(* IEC 61131-3 sources: simulador/simulador_codesys, 11 files *)

(* ---- GVL_SimConfig.st ---- *)
// =============================================================================
// GVL_SimConfig — Parâmetros globais de configuração do simulador
// Equivalente a: config.py + config_etapa1/2/3.yaml
//
// COMO USAR:
//   Etapa 1 (loopback)  → SIM_MODE := 0
//   Etapa 2 (openloop)  → SIM_MODE := 1
//   Etapa 3 (full)      → SIM_MODE := 2
//
// Alterar SIM_MODE em tempo de execução reinicializa o comportamento na
// próxima chamada de FB_Simulator (bEdgeInit detecta a mudança).
// =============================================================================

VAR_GLOBAL CONSTANT

    // -------------------------------------------------------------------------
    // Modo de simulação
    //   0 = LOOPBACK  — comunicação Modbus, medidor fixo, física OFF
    //   1 = OPENLOOP  — física ON, carga/irradiância fixas, sem perfis/eventos
    //   2 = FULL      — física ON, perfis ativos, eventos ativos
    // -------------------------------------------------------------------------
    SIM_MODE_LOOPBACK   : INT := 0;
    SIM_MODE_OPENLOOP   : INT := 1;
    SIM_MODE_FULL       : INT := 2;

    // -------------------------------------------------------------------------
    // Temporização
    // -------------------------------------------------------------------------
    TICK_S              : REAL := 0.05;     // Período do ciclo de simulação (s)
                                             // Deve coincidir com o período da
                                             // task cíclica no Codesys Scheduler.
                                             // 50 ms é o mínimo seguro.

    // -------------------------------------------------------------------------
    // Rede elétrica
    // -------------------------------------------------------------------------
    V_LL_V              : REAL := 380.0;    // Tensão nominal linha-linha BT (V)
    V_MT_LL_V           : REAL := 13800.0;  // Tensão nominal linha-linha MT (V)

    // -------------------------------------------------------------------------
    // Equivalente de Thévenin da rede (referido ao BT)
    // -------------------------------------------------------------------------
    THEVENIN_VTH_LL_V   : REAL := 380.0;   // Tensão de Thévenin LL (V)
    THEVENIN_R_OHM      : REAL := 0.00283; // Resistência equivalente (Ω)
    THEVENIN_X_OHM      : REAL := 0.01416; // Reatância equivalente (Ω)

    // -------------------------------------------------------------------------
    // Relações de transformação dos instrumentos
    // -------------------------------------------------------------------------
    RTP                 : REAL := 120.0;    // Relação do TP  (ex: 13800/115 → 120)
    RTC                 : REAL := 200.0;    // Relação do TC  (ex: 200/5 → 200)

    // -------------------------------------------------------------------------
    // Modelo de carga ZIP (coeficientes ANEEL para alimentadores)
    //   P: 50% impedância constante + 50% potência constante
    //   Q: 100% potência constante
    // -------------------------------------------------------------------------
    ZIP_P_Z             : REAL := 0.50;    // Fração Z para P
    ZIP_P_I             : REAL := 0.00;    // Fração I para P
    ZIP_P_P             : REAL := 0.50;    // Fração P para P
    ZIP_Q_Z             : REAL := 0.00;    // Fração Z para Q
    ZIP_Q_I             : REAL := 0.00;    // Fração I para Q
    ZIP_Q_P             : REAL := 1.00;    // Fração P para Q

    // -------------------------------------------------------------------------
    // Carga padrão (usada em openloop e como fallback no full)
    // -------------------------------------------------------------------------
    LOAD_P_KW_DEFAULT   : REAL := 200.0;   // Potência ativa da carga (kW)
    LOAD_Q_KVAR_DEFAULT : REAL := 50.0;    // Potência reativa da carga (kVAr)

    // -------------------------------------------------------------------------
    // Irradiância padrão (normalizada 0.0..1.0)
    // -------------------------------------------------------------------------
    U_DEFAULT           : REAL := 1.0;     // 1.0 = irradiância plena (100%)

    // -------------------------------------------------------------------------
    // Valores fixos do medidor no modo LOOPBACK (grandezas no SECUNDÁRIO)
    //   V_sec_fn = V_MT_fn / RTP = (13800 / sqrt(3)) / 120 ≈ 66.4 V
    //   I_sec    = valor de teste no secundário do TC
    //   PF       = fator de potência de teste
    // -------------------------------------------------------------------------
    LOOPBACK_PF         : REAL := 0.92;    // Fator de potência fixo (loopback)
    LOOPBACK_V_MT_LN_V  : REAL := 66.4;   // Tensão sec. TP fase-neutro (V)
    LOOPBACK_I_MT_A     : REAL := 2.5;    // Corrente sec. TC (A)

    // -------------------------------------------------------------------------
    // Medidor Modbus (slave 100, COM1)
    // -------------------------------------------------------------------------
    METER_SLAVE_ID      : INT  := 100;
    METER_BASE_ADDR     : INT  := 153;     // 0x0099 decimal — endereço base FC03
    METER_QTY_U16       : INT  := 28;      // Quantidade de registradores U16

    // -------------------------------------------------------------------------
    // Número total de inversores
    //   COM1: slaves 101..109  (9 inversores)
    //   COM2: slaves 201..209  (9 inversores)
    // -------------------------------------------------------------------------
    N_INV               : INT  := 18;      // Total de inversores
    N_INV_COM1          : INT  := 9;       // Inversores na COM1 (índices 0..8)
    N_INV_COM2          : INT  := 9;       // Inversores na COM2 (índices 9..17)

    // -------------------------------------------------------------------------
    // Slave IDs dos inversores
    //   Índice 0..8  → COM1: slaves 101..109
    //   Índice 9..17 → COM2: slaves 201..209
    // -------------------------------------------------------------------------
    INV_SLAVE_ID        : ARRAY[0..17] OF INT := [
        101, 102, 103, 104, 105, 106, 107, 108, 109,   // COM1
        201, 202, 203, 204, 205, 206, 207, 208, 209    // COM2
    ];

    // -------------------------------------------------------------------------
    // Potências nominais dos inversores (kW)
    // -------------------------------------------------------------------------
    INV_P_NOM_KW        : ARRAY[0..17] OF REAL := [
        60.0, 60.0, 35.0, 15.0, 15.0, 15.0, 15.0, 15.0, 15.0,  // COM1
        15.0, 15.0, 15.0, 15.0, 15.0, 15.0, 35.0, 35.0, 50.0   // COM2
    ];

    // -------------------------------------------------------------------------
    // Potências aparentes nominais dos inversores (kVA)
    // -------------------------------------------------------------------------
    INV_S_NOM_KVA       : ARRAY[0..17] OF REAL := [
        60.0, 60.0, 35.0, 15.0, 15.0, 15.0, 15.0, 15.0, 15.0,  // COM1
        15.0, 15.0, 15.0, 15.0, 15.0, 15.0, 35.0, 35.0, 50.0   // COM2
    ];

    // -------------------------------------------------------------------------
    // Constantes de tempo dos inversores (s)
    //   tau_p: dinâmica de P (1ª ordem)
    //   tau_q: dinâmica de Q (1ª ordem)
    // -------------------------------------------------------------------------
    INV_TAU_P_S         : ARRAY[0..17] OF REAL := [
        1.0, 1.0, 1.0, 1.0, 1.0, 1.0, 1.0, 1.0, 1.0,
        1.0, 1.0, 1.0, 1.0, 1.0, 1.0, 1.0, 1.0, 1.0
    ];
    INV_TAU_Q_S         : ARRAY[0..17] OF REAL := [
        1.0, 1.0, 1.0, 1.0, 1.0, 1.0, 1.0, 1.0, 1.0,
        1.0, 1.0, 1.0, 1.0, 1.0, 1.0, 1.0, 1.0, 1.0
    ];

    // -------------------------------------------------------------------------
    // Endereços Modbus dos inversores (Holding Registers, base 0)
    // -------------------------------------------------------------------------
    INV_HR_P_PCT        : INT := 256;      // HR 256 → setpoint %P  (escrito pelo master)
    INV_HR_PF_RAW       : INT := 257;      // HR 257 → FP raw       (escrito pelo master)

    // -------------------------------------------------------------------------
    // Eventos: intervalo de releitura (s)
    // -------------------------------------------------------------------------
    EVENTS_POLL_S       : REAL := 2.0;

END_VAR

(* ---- GVL_SimState.st ---- *)
// =============================================================================
// GVL_SimState — Estado em tempo de execução do simulador
// Equivalente às dataclasses InverterState, MeterState e PlantSimulation
// em simulation.py.
//
// Estas variáveis são LIDAS/ESCRITAS pelo FB_Simulator a cada ciclo.
// O driver Modbus Slave do Codesys mapeia diretamente os registradores
// do medidor (MW_Meter) e dos inversores (MW_Inv_*) em memória.
// =============================================================================

VAR_GLOBAL

    // =========================================================================
    // CONTROLE GERAL
    // =========================================================================

    // Modo ativo (alterável em runtime via HMI ou variável)
    //   0 = LOOPBACK | 1 = OPENLOOP | 2 = FULL
    g_SimMode           : INT := 0;

    // Tempo acumulado de simulação (s) — avança a cada ciclo
    g_T_s               : REAL := 0.0;

    // Flag de reinicialização: setar TRUE para reiniciar estados
    g_Reset             : BOOL := FALSE;

    // =========================================================================
    // ESTADO DOS INVERSORES
    // =========================================================================

    // --- Setpoints recebidos do master via FC16 (escritos pelo driver Modbus) ---
    // HR 256: setpoint %P  (0..100)
    g_Inv_P_Ref_Pct     : ARRAY[0..17] OF REAL := [18(0.0)];

    // HR 257: FP raw (1..100)
    g_Inv_PF_Cmd_Raw    : ARRAY[0..17] OF INT  := [18(100)];

    // --- Estados internos da dinâmica de 1ª ordem ---
    g_Inv_P_kW          : ARRAY[0..17] OF REAL := [18(0.0)];
    g_Inv_Q_kVAr        : ARRAY[0..17] OF REAL := [18(0.0)];

    // --- Disponibilidade de energia (irradiância normalizada 0..1) ---
    g_Inv_U             : ARRAY[0..17] OF REAL := [18(1.0)];

    // --- Flags de eventos ---
    g_Inv_CommsDrop     : ARRAY[0..17] OF BOOL := [18(FALSE)];
    g_Inv_Frozen_s      : ARRAY[0..17] OF REAL := [18(0.0)];

    // =========================================================================
    // ESTADO DO MEDIDOR (grandezas no SECUNDÁRIO dos instrumentos)
    // =========================================================================
    // O driver Modbus Slave mapeia MW_Meter[] nos registradores FC03
    // a partir do endereço base 0x0099 (153 decimal).
    // Cada elemento é um UINT (U16) codificado conforme especificação.

    // Registradores raw U16 para o driver Modbus Slave
    // Índice 0..27 → offsets relativos a 0x0099
    //   [0]  = PF fase A     [1]  = PF fase B     [2]  = PF fase C
    //   [3..6] = reservado = 0
    //   [7]  = Ia sec        [8]  = Ib sec         [9]  = Ic sec
    //   [10] = reservado = 0
    //   [11] = Ua sec fn     [12] = Ub sec fn      [13] = Uc sec fn
    //   [14..27] = reservado = 0
    MW_Meter            : ARRAY[0..27] OF UINT := [28(0)];

    // Grandezas físicas internas do medidor (REAL, para debug/HMI)
    g_Meter_PFa         : REAL := 1.0;
    g_Meter_PFb         : REAL := 1.0;
    g_Meter_PFc         : REAL := 1.0;
    g_Meter_Ia_A        : REAL := 0.0;  // corrente sec. TC (A)
    g_Meter_Ib_A        : REAL := 0.0;
    g_Meter_Ic_A        : REAL := 0.0;
    g_Meter_Ua_V        : REAL := 0.0;  // tensão sec. TP fase-neutro (V)
    g_Meter_Ub_V        : REAL := 0.0;
    g_Meter_Uc_V        : REAL := 0.0;
    g_Meter_P_PCC_kW    : REAL := 0.0;  // potência ativa no PCC (kW)
    g_Meter_Q_PCC_kVAr  : REAL := 0.0;  // potência reativa no PCC (kVAr)
    g_Meter_V_PCC_LL_V  : REAL := 380.0; // tensão linha-linha no PCC (V)

    // =========================================================================
    // EVENTOS EM TEMPO REAL (equivalente a events.json)
    // Alteráveis via HMI Codesys ou CoDeSys VisualizationControl
    // =========================================================================

    // drop_comms: TRUE = inversor perde comunicação (rampa P→0 em 5 s)
    g_Ev_DropComms      : ARRAY[0..17] OF BOOL := [18(FALSE)];

    // freeze_s: segundos restantes de congelamento de firmware (0 = normal)
    g_Ev_Freeze_s       : ARRAY[0..17] OF REAL := [18(0.0)];

    // force_u: sobrescreve irradiância do inversor (−1 = não forçar)
    //   −1.0 = usa u_global do perfil
    //   0.0..1.0 = força esta irradiância (sombreamento)
    g_Ev_Force_U        : ARRAY[0..17] OF REAL := [18(-1.0)];

    // =========================================================================
    // PERFIS (equivalente a u_profile.csv e load_profile.csv)
    // Piecewise-constant: valor vira ativo quando g_T_s >= time_s[i]
    // =========================================================================

    // --- Perfil de irradiância (u_profile.csv) ---
    // Dimensione conforme o número de pontos do seu perfil (máx. 64 pontos)
    U_PROFILE_N         : INT := 5;        // Número de pontos ativos
    U_Profile_T_s       : ARRAY[0..63] OF DINT := [
          0,   300,   600,   900,  1200,
         59(0)
    ];
    U_Profile_Val       : ARRAY[0..63] OF REAL := [
        1.0,   0.7,   0.4,   0.8,   1.0,
        59(0.0)
    ];

    // --- Perfil de carga (load_profile.csv) ---
    LOAD_PROFILE_N      : INT := 5;
    Load_Profile_T_s    : ARRAY[0..63] OF DINT := [
          0,   300,   600,   900,  1200,
         59(0)
    ];
    Load_Profile_P_kW   : ARRAY[0..63] OF REAL := [
        200.0, 250.0, 180.0, 220.0, 200.0,
        59(0.0)
    ];
    Load_Profile_Q_kVAr : ARRAY[0..63] OF REAL := [
         50.0,  60.0,  45.0,  55.0,  50.0,
         59(0.0)
    ];

    // =========================================================================
    // DIAGNÓSTICO
    // =========================================================================
    g_P_Gen_Total_kW    : REAL := 0.0;   // Soma P de todos inversores
    g_Q_Gen_Total_kVAr  : REAL := 0.0;   // Soma Q de todos inversores
    g_CycleOverrun      : BOOL := FALSE; // TRUE se task demorou mais que TICK_S

END_VAR

(* ---- FC_DecodePF.st ---- *)
// =============================================================================
// FC_DecodePF — Decodifica FP raw (U16) enviado pelo master ao inversor
// Equivalente a PlantSimulation._decode_pf() em simulation.py
//
// Protocolo:
//   1..20   → lagging (indutivo):  PF = 1.00 − raw×0.01    (0.80..0.99)
//             sign_q = −1  →  Q < 0  (consome reativo)
//   80..99  → leading (capacitivo): PF = raw/100            (0.80..0.99)
//             sign_q = +1  →  Q > 0  (injeta reativo)
//   100     → unitário: PF = 1.0, Q = 0
//   21..79  → inválido: tratado como unitário
//
// Saídas:
//   pf_mag  : REAL  — magnitude do FP (0.80..1.00)
//   sign_q  : INT   — +1 leading | −1 lagging | 0 unitário
// =============================================================================

FUNCTION FC_DecodePF : BOOL    // retorna TRUE sempre (função não falha)
VAR_INPUT
    raw     : INT;              // FP raw recebido via HR 257
END_VAR
VAR_OUTPUT
    pf_mag  : REAL;             // Magnitude do FP
    sign_q  : INT;              // Sinal de Q: +1 | 0 | -1
END_VAR

IF raw >= 1 AND raw <= 20 THEN
    // Lagging (indutivo): consome reativo, Q < 0
    pf_mag := 1.0 - REAL(raw) * 0.01;
    IF pf_mag < 0.80 THEN pf_mag := 0.80; END_IF
    IF pf_mag > 0.99 THEN pf_mag := 0.99; END_IF
    sign_q := -1;

ELSIF raw >= 80 AND raw <= 99 THEN
    // Leading (capacitivo): injeta reativo, Q > 0
    pf_mag := REAL(raw) / 100.0;
    IF pf_mag < 0.80 THEN pf_mag := 0.80; END_IF
    IF pf_mag > 0.99 THEN pf_mag := 0.99; END_IF
    sign_q := 1;

ELSIF raw = 100 THEN
    // Unitário
    pf_mag := 1.0;
    sign_q := 0;

ELSE
    // Fora de faixa (21..79 ou negativo) → trata como unitário
    pf_mag := 1.0;
    sign_q := 0;
END_IF

FC_DecodePF := TRUE;

END_FUNCTION

(* ---- FC_EncodeIV.st ---- *)
// =============================================================================
// FC_EncodeI — Codifica corrente secundária TC em UINT (U16)
// Equivalente a modbus_server.py → encode_i_u16()
//
// Resolução: 1/256 A por LSB
//   reg = ROUND(I_sec_A × 256)
//   Master reconstrói: I_sec = reg / 256
//   I_prim = I_sec × RTC
// =============================================================================

FUNCTION FC_EncodeI : UINT
VAR_INPUT
    i_a : REAL;     // Corrente secundária TC (A), ≥ 0
END_VAR
VAR
    raw : DINT;
END_VAR

IF i_a < 0.0 THEN i_a := 0.0; END_IF
raw := REAL_TO_DINT(i_a * 256.0 + 0.5);
IF raw > 65535 THEN raw := 65535; END_IF
FC_EncodeI := DINT_TO_UINT(raw);

END_FUNCTION

// =============================================================================
// FC_EncodeV — Codifica tensão secundária TP em UINT (U16)
// Equivalente a modbus_server.py → encode_v_u16()
//
// Resolução: 1/128 V por LSB
//   reg = ROUND(V_sec_V × 128)
//   Master reconstrói: V_sec = reg / 128
//   V_prim = V_sec × RTP
// =============================================================================

FUNCTION FC_EncodeV : UINT
VAR_INPUT
    v_v : REAL;     // Tensão secundária TP fase-neutro (V), ≥ 0
END_VAR
VAR
    raw : DINT;
END_VAR

IF v_v < 0.0 THEN v_v := 0.0; END_IF
raw := REAL_TO_DINT(v_v * 128.0 + 0.5);
IF raw > 65535 THEN raw := 65535; END_IF
FC_EncodeV := DINT_TO_UINT(raw);

END_FUNCTION

(* ---- FC_EncodePF.st ---- *)
// =============================================================================
// FC_EncodePF — Codifica fator de potência com sinal em UINT (U16)
// Equivalente a modbus_server.py → encode_pf_u16()
//
// Convenção (igual ao Python):
//   pf ∈ [ 0.0,  1.0] → reg = ROUND(pf × 16384)         (0..16384)
//   pf ∈ [-1.0,  0.0) → reg = 65535 − ROUND(|pf| × 16384)
//
// O master (WAGO SCRPI) decodifica:
//   se reg ≤ 16384  → pf =  reg / 16384
//   se reg ≥ 49151  → pf = -(65535 - reg) / 16384
// =============================================================================

FUNCTION FC_EncodePF : UINT
VAR_INPUT
    pf  : REAL;     // Fator de potência com sinal (−1.0 .. +1.0)
END_VAR
VAR
    pf_sat  : REAL;
    raw     : DINT;
END_VAR

// Saturar entrada
pf_sat := pf;
IF pf_sat >  1.0 THEN pf_sat :=  1.0; END_IF
IF pf_sat < -1.0 THEN pf_sat := -1.0; END_IF

IF pf_sat >= 0.0 THEN
    // Positivo: indutivo (Q > 0)
    raw := REAL_TO_DINT(pf_sat * 16384.0 + 0.5);   // arredondamento
    IF raw > 16384 THEN raw := 16384; END_IF
    FC_EncodePF := DINT_TO_UINT(raw);
ELSE
    // Negativo: capacitivo (Q < 0)
    raw := REAL_TO_DINT(ABS(pf_sat) * 16384.0 + 0.5);
    IF raw > 16384 THEN raw := 16384; END_IF
    FC_EncodePF := DINT_TO_UINT(65535 - raw);
END_IF

END_FUNCTION

(* ---- FC_ProfileStep.st ---- *)
// =============================================================================
// FC_ProfileStep — Leitura de perfil piecewise-constant (step profile)
// Equivalente a profiles.py → StepProfile.value()
//
// O valor vigente é o último ponto com T_s[i] <= t_s.
// Se nenhum ponto for atingido, retorna default_val.
//
// Uso para perfil de irradiância (u_profile):
//   u := FC_ProfileStep(
//       t_s         := REAL_TO_DINT(g_T_s),
//       n           := U_PROFILE_N,
//       T_s         := U_Profile_T_s,
//       vals        := U_Profile_Val,
//       default_val := U_DEFAULT
//   );
//
// Uso para perfil de carga: chamar 2x (uma para P, outra para Q),
//   passando Load_Profile_P_kW ou Load_Profile_Q_kVAr como vals.
// =============================================================================

FUNCTION FC_ProfileStep : REAL
VAR_INPUT
    t_s         : DINT;                     // Tempo atual (s, inteiro)
    n           : INT;                      // Número de pontos ativos
    T_s         : ARRAY[0..63] OF DINT;    // Tempos dos pontos (s)
    vals        : ARRAY[0..63] OF REAL;    // Valores nos pontos
    default_val : REAL;                     // Valor se nenhum ponto atingido
END_VAR
VAR
    i       : INT;
    result  : REAL;
END_VAR

result := default_val;

FOR i := 0 TO n - 1 DO
    IF t_s >= T_s[i] THEN
        result := vals[i];
    ELSE
        EXIT;   // Lista ordenada: pode parar no primeiro ponto futuro
    END_IF
END_FOR

FC_ProfileStep := result;

END_FUNCTION

(* ---- FB_InverterDyn.st ---- *)
// =============================================================================
// FB_InverterDyn — Dinâmica de 1ª ordem de um inversor fotovoltaico
// Equivalente ao loop de inversores em PlantSimulation.step()
//
// Modela um inversor como dois filtros de 1ª ordem independentes (P e Q),
// com saturação na potência disponível (u × P_nom) e no limite de S_nom.
//
// Discretização: Euler explícito
//   P[k+1] = P[k] + (Ts/tau_p) × (P_ref − P[k])
//   Q[k+1] = Q[k] + (Ts/tau_q) × (Q_ref − Q[k])
//
// Um bloco FB_InverterDyn é instanciado para cada inversor (0..17).
// O FB_Simulator chama todos a cada ciclo.
// =============================================================================

FUNCTION_BLOCK FB_InverterDyn
VAR_INPUT
    // Parâmetros fixos (configurados uma vez)
    p_nom_kw    : REAL;     // Potência ativa nominal (kW)
    s_nom_kva   : REAL;     // Potência aparente nominal (kVA)
    tau_p_s     : REAL;     // Constante de tempo de P (s)
    tau_q_s     : REAL;     // Constante de tempo de Q (s)
    tick_s      : REAL;     // Período de amostragem (s) = TICK_S

    // Setpoints (escritos pelo driver Modbus a cada FC16)
    p_ref_pct   : REAL;     // Setpoint %P  (0..100)
    pf_cmd_raw  : INT;      // FP raw HR257 (1..100)

    // Disponibilidade de energia (irradiância normalizada 0..1)
    u           : REAL;

    // Eventos
    comms_drop  : BOOL;     // TRUE = perda de comunicação (rampa P→0)
    frozen_s    : REAL;     // Segundos restantes de congelamento
END_VAR
VAR_OUTPUT
    p_kw        : REAL;     // Potência ativa atual (kW)
    q_kvar      : REAL;     // Potência reativa atual (kVAr)
    frozen_s_out: REAL;     // Tempo de congelamento restante após step
    p_ref_pct_out: REAL;    // p_ref_pct após aplicação de drop_comms
END_VAR
VAR
    alpha       : REAL;     // Ts / tau_p
    beta        : REAL;     // Ts / tau_q
    p_avail     : REAL;     // Potência disponível (u × p_nom)
    p_ref_kw    : REAL;     // Referência de P em kW
    pf_mag      : REAL;
    sign_q      : INT;
    q_ref       : REAL;
    q_lim       : REAL;
    q_lim_sq    : REAL;
    p_ref_pct_w : REAL;     // cópia de trabalho de p_ref_pct
    SQRT3       : REAL := 1.7320508;
    COS_INV_ARG : REAL;
    // variáveis internas de estado (persistem entre chamadas)
    _p_kw       : REAL;
    _q_kvar     : REAL;
END_VAR

// -----------------------------------------------------------------------
// Preservar saídas com estado persistente
// -----------------------------------------------------------------------
p_kw  := _p_kw;
q_kvar := _q_kvar;

// -----------------------------------------------------------------------
// Congelamento de firmware: P e Q ficam constantes, decrementar timer
// -----------------------------------------------------------------------
IF frozen_s > 0.0 THEN
    frozen_s_out  := frozen_s - tick_s;
    IF frozen_s_out < 0.0 THEN frozen_s_out := 0.0; END_IF
    p_ref_pct_out := p_ref_pct;
    // P e Q NÃO mudam — retornar valores atuais
    RETURN;
END_IF
frozen_s_out := 0.0;

// -----------------------------------------------------------------------
// Perda de comunicação: rampa P a zero em 5 s
// -----------------------------------------------------------------------
p_ref_pct_w := p_ref_pct;
IF comms_drop THEN
    p_ref_pct_w := p_ref_pct_w - (tick_s / 5.0) * 100.0;
    IF p_ref_pct_w < 0.0 THEN p_ref_pct_w := 0.0; END_IF
END_IF
p_ref_pct_out := p_ref_pct_w;

// -----------------------------------------------------------------------
// Constantes de tempo discretizadas (Euler explícito)
// -----------------------------------------------------------------------
IF tau_p_s > 0.0 THEN
    alpha := tick_s / tau_p_s;
ELSE
    alpha := 1.0;
END_IF

IF tau_q_s > 0.0 THEN
    beta := tick_s / tau_q_s;
ELSE
    beta := 1.0;
END_IF

// Saturar alpha/beta em 1.0 para evitar instabilidade numérica
IF alpha > 1.0 THEN alpha := 1.0; END_IF
IF beta  > 1.0 THEN beta  := 1.0; END_IF

// -----------------------------------------------------------------------
// Potência ativa
// -----------------------------------------------------------------------
p_avail  := u * p_nom_kw;
IF p_avail < 0.0 THEN p_avail := 0.0; END_IF

p_ref_kw := (p_ref_pct_w / 100.0) * p_nom_kw;

_p_kw := _p_kw + alpha * (p_ref_kw - _p_kw);

// Saturar em [0, p_avail]
IF _p_kw < 0.0     THEN _p_kw := 0.0;     END_IF
IF _p_kw > p_avail THEN _p_kw := p_avail; END_IF

// -----------------------------------------------------------------------
// Potência reativa — decodifica FP raw e calcula Q_ref
// -----------------------------------------------------------------------
FC_DecodePF(raw := pf_cmd_raw, pf_mag => pf_mag, sign_q => sign_q);

IF pf_mag >= 0.9999 OR sign_q = 0 THEN
    q_ref := 0.0;
ELSE
    // Q_ref = sign_q × P × tan(acos(pf_mag))
    // Usando identidade: tan(acos(x)) = sqrt(1-x²)/x
    COS_INV_ARG := 1.0 - pf_mag * pf_mag;
    IF COS_INV_ARG < 0.0 THEN COS_INV_ARG := 0.0; END_IF
    q_ref := REAL(sign_q) * _p_kw * SQRT(COS_INV_ARG) / pf_mag;
END_IF

// Limite de Q pela capacidade aparente: |Q| ≤ sqrt(S² − P²)
q_lim_sq := s_nom_kva * s_nom_kva - _p_kw * _p_kw;
IF q_lim_sq < 0.0 THEN q_lim_sq := 0.0; END_IF
q_lim := SQRT(q_lim_sq);

_q_kvar := _q_kvar + beta * (q_ref - _q_kvar);

// Saturar em [−q_lim, +q_lim]
IF _q_kvar < -q_lim THEN _q_kvar := -q_lim; END_IF
IF _q_kvar >  q_lim THEN _q_kvar :=  q_lim; END_IF

// -----------------------------------------------------------------------
// Atualizar saídas com estado persistente
// -----------------------------------------------------------------------
p_kw   := _p_kw;
q_kvar := _q_kvar;

END_FUNCTION_BLOCK

(* ---- FB_Simulator.st ---- *)
// =============================================================================
// FB_Simulator — Bloco principal do simulador de usina FV
// Equivalente a PlantSimulation (simulation.py) + main.py
//
// Chamado ciclicamente pela task de simulação (período = TICK_S).
// Lê setpoints de g_Inv_P_Ref_Pct[] e g_Inv_PF_Cmd_Raw[] (escritos pelo
// driver Modbus Slave quando o master envia FC16).
// Escreve MW_Meter[] (lido pelo driver Modbus Slave para responder FC03).
//
// MODOS (g_SimMode):
//   SIM_MODE_LOOPBACK (0) — medidor fixo, sem física
//   SIM_MODE_OPENLOOP (1) — física ativa, carga/u fixas
//   SIM_MODE_FULL     (2) — física + perfis + eventos
//
// RESET:
//   Setar g_Reset := TRUE para zerar todos os estados dinâmicos.
//   O FB limpa g_Reset automaticamente após reset.
// =============================================================================

FUNCTION_BLOCK FB_Simulator
VAR_INPUT
    // Sem entradas externas — tudo via GVL_SimState e GVL_SimConfig
END_VAR
VAR_OUTPUT
    // Sem saídas diretas — escreve nas GVLs
END_VAR
VAR
    // -----------------------------------------------------------------------
    // Instâncias dos modelos físicos
    // -----------------------------------------------------------------------
    fbThevenin  : FB_Thevenin;
    fbZipLoad   : FB_ZipLoad;
    fbInv       : ARRAY[0..17] OF FB_InverterDyn;

    // -----------------------------------------------------------------------
    // Variáveis de trabalho internas
    // -----------------------------------------------------------------------
    i               : INT;
    t_int           : DINT;

    // Carga
    load_p0_kw      : REAL;
    load_q0_kvar    : REAL;
    load_p_kw       : REAL;
    load_q_kvar     : REAL;

    // Irradiância global
    u_global        : REAL;
    u_inv           : REAL;

    // PCC 1ª iteração
    p_gen           : REAL;
    q_gen           : REAL;
    p_pcc_0         : REAL;
    q_pcc_0         : REAL;
    v_pcc_0         : REAL;

    // PCC 2ª iteração
    p_pcc           : REAL;
    q_pcc           : REAL;
    s_pcc           : REAL;
    s_pcc_sq        : REAL;
    v_pcc_ll        : REAL;

    // Medidor — grandezas calculadas
    pf_mag          : REAL;
    pf_signed       : REAL;
    v_pcc_fn        : REAL;
    v_mt_fn         : REAL;
    v_mt_ll         : REAL;
    v_sec_fn        : REAL;
    i_mt_prim       : REAL;
    i_sec           : REAL;

    // Controle de modo anterior (detecta mudança de modo)
    _prev_mode      : INT := -1;

    // Constantes matemáticas
    SQRT3           : REAL := 1.7320508;
    SQRT3_INV       : REAL := 0.5773503;    // 1/sqrt(3)

    // Evento drop_comms: cópia de p_ref_pct após aplicação da rampa
    _p_ref_pct_eff  : ARRAY[0..17] OF REAL;
END_VAR

// ===========================================================================
// RESET
// ===========================================================================
IF g_Reset THEN
    g_T_s := 0.0;
    FOR i := 0 TO 17 DO
        g_Inv_P_kW[i]      := 0.0;
        g_Inv_Q_kVAr[i]    := 0.0;
        g_Inv_U[i]         := 1.0;
        g_Inv_CommsDrop[i] := FALSE;
        g_Inv_Frozen_s[i]  := 0.0;
        // Zerar estados internos dos FB de inversores via re-init
        // (no Codesys, reinicializar instâncias de FB não é direto;
        //  o workaround é forçar p_kw=0 via setpoint zero e esperar decaimento,
        //  ou usar o campo _p_kw diretamente se a versão do Codesys permitir.)
        g_Inv_P_Ref_Pct[i]  := 0.0;
        g_Inv_PF_Cmd_Raw[i] := 100;
    END_FOR
    g_Meter_P_PCC_kW    := 0.0;
    g_Meter_Q_PCC_kVAr  := 0.0;
    g_Meter_V_PCC_LL_V  := V_LL_V;
    _prev_mode          := -1;
    g_Reset             := FALSE;
    RETURN;
END_IF

// ===========================================================================
// DETECÇÃO DE MUDANÇA DE MODO
// ===========================================================================
IF g_SimMode <> _prev_mode THEN
    _prev_mode := g_SimMode;
    // Ao entrar no modo LOOPBACK: inicializa medidor com valores fixos
    IF g_SimMode = SIM_MODE_LOOPBACK THEN
        g_Meter_PFa := LOOPBACK_PF;
        g_Meter_PFb := LOOPBACK_PF;
        g_Meter_PFc := LOOPBACK_PF;
        g_Meter_Ia_A := LOOPBACK_I_MT_A;
        g_Meter_Ib_A := LOOPBACK_I_MT_A;
        g_Meter_Ic_A := LOOPBACK_I_MT_A;
        g_Meter_Ua_V := LOOPBACK_V_MT_LN_V;
        g_Meter_Ub_V := LOOPBACK_V_MT_LN_V;
        g_Meter_Uc_V := LOOPBACK_V_MT_LN_V;
        // Codifica e preenche MW_Meter
        MW_Meter[0]  := FC_EncodePF(LOOPBACK_PF);
        MW_Meter[1]  := FC_EncodePF(LOOPBACK_PF);
        MW_Meter[2]  := FC_EncodePF(LOOPBACK_PF);
        MW_Meter[3]  := 0;  MW_Meter[4]  := 0;
        MW_Meter[5]  := 0;  MW_Meter[6]  := 0;
        MW_Meter[7]  := FC_EncodeI(LOOPBACK_I_MT_A);
        MW_Meter[8]  := FC_EncodeI(LOOPBACK_I_MT_A);
        MW_Meter[9]  := FC_EncodeI(LOOPBACK_I_MT_A);
        MW_Meter[10] := 0;
        MW_Meter[11] := FC_EncodeV(LOOPBACK_V_MT_LN_V);
        MW_Meter[12] := FC_EncodeV(LOOPBACK_V_MT_LN_V);
        MW_Meter[13] := FC_EncodeV(LOOPBACK_V_MT_LN_V);
        MW_Meter[14] := 0;  MW_Meter[15] := 0;  MW_Meter[16] := 0;
        MW_Meter[17] := 0;  MW_Meter[18] := 0;  MW_Meter[19] := 0;
        MW_Meter[20] := 0;  MW_Meter[21] := 0;  MW_Meter[22] := 0;
        MW_Meter[23] := 0;  MW_Meter[24] := 0;  MW_Meter[25] := 0;
        MW_Meter[26] := 0;  MW_Meter[27] := 0;
    END_IF
END_IF

// ===========================================================================
// AVANÇA TEMPO
// ===========================================================================
g_T_s := g_T_s + TICK_S;
t_int := REAL_TO_DINT(g_T_s);

// ===========================================================================
// MODO LOOPBACK — sem física, apenas loga setpoints recebidos
// ===========================================================================
IF g_SimMode = SIM_MODE_LOOPBACK THEN
    // MW_Meter já foi preenchido na detecção de mudança de modo.
    // Inversores apenas registram o que o master enviou (sem simulação).
    // (O log seria feito via variável de diagnóstico em HMI)
    RETURN;
END_IF

// ===========================================================================
// MODOS OPENLOOP e FULL — física ativa
// ===========================================================================

// ---------------------------------------------------------------------------
// 1. Perfis de irradiância e carga
// ---------------------------------------------------------------------------
IF g_SimMode = SIM_MODE_FULL THEN
    u_global := FC_ProfileStep(
        t_s         := t_int,
        n           := U_PROFILE_N,
        T_s         := U_Profile_T_s,
        vals        := U_Profile_Val,
        default_val := U_DEFAULT
    );
    IF u_global < 0.0 THEN u_global := 0.0; END_IF
    IF u_global > 1.0 THEN u_global := 1.0; END_IF

    load_p0_kw := FC_ProfileStep(
        t_s         := t_int,
        n           := LOAD_PROFILE_N,
        T_s         := Load_Profile_T_s,
        vals        := Load_Profile_P_kW,
        default_val := LOAD_P_KW_DEFAULT
    );
    load_q0_kvar := FC_ProfileStep(
        t_s         := t_int,
        n           := LOAD_PROFILE_N,
        T_s         := Load_Profile_T_s,
        vals        := Load_Profile_Q_kVAr,
        default_val := LOAD_Q_KVAR_DEFAULT
    );
ELSE
    // OPENLOOP: valores fixos do YAML / GVL_SimConfig
    u_global     := U_DEFAULT;
    IF u_global < 0.0 THEN u_global := 0.0; END_IF
    IF u_global > 1.0 THEN u_global := 1.0; END_IF
    load_p0_kw   := LOAD_P_KW_DEFAULT;
    load_q0_kvar := LOAD_Q_KVAR_DEFAULT;
END_IF

// ---------------------------------------------------------------------------
// 2. Dinâmica de cada inversor
// ---------------------------------------------------------------------------
FOR i := 0 TO 17 DO

    // Disponibilidade de energia (irradiância por inversor)
    IF g_SimMode = SIM_MODE_FULL AND g_Ev_Force_U[i] >= 0.0 THEN
        u_inv := g_Ev_Force_U[i];
        IF u_inv > 1.0 THEN u_inv := 1.0; END_IF
    ELSE
        u_inv := u_global;
    END_IF
    g_Inv_U[i] := u_inv;

    // drop_comms: só no modo full
    IF g_SimMode = SIM_MODE_FULL THEN
        g_Inv_CommsDrop[i] := g_Ev_DropComms[i];
    ELSE
        g_Inv_CommsDrop[i] := FALSE;
    END_IF

    // freeze_s: só no modo full; acumulativo — usa o maior valor entre restante e evento
    IF g_SimMode = SIM_MODE_FULL THEN
        IF g_Ev_Freeze_s[i] > g_Inv_Frozen_s[i] THEN
            g_Inv_Frozen_s[i] := g_Ev_Freeze_s[i];
        END_IF
    END_IF

    // Chamar FB de dinâmica do inversor
    fbInv[i](
        p_nom_kw      := INV_P_NOM_KW[i],
        s_nom_kva     := INV_S_NOM_KVA[i],
        tau_p_s       := INV_TAU_P_S[i],
        tau_q_s       := INV_TAU_Q_S[i],
        tick_s        := TICK_S,
        p_ref_pct     := g_Inv_P_Ref_Pct[i],
        pf_cmd_raw    := g_Inv_PF_Cmd_Raw[i],
        u             := u_inv,
        comms_drop    := g_Inv_CommsDrop[i],
        frozen_s      := g_Inv_Frozen_s[i]
    );

    // Realimentar estados e saídas do FB
    g_Inv_P_kW[i]     := fbInv[i].p_kw;
    g_Inv_Q_kVAr[i]   := fbInv[i].q_kvar;
    g_Inv_Frozen_s[i] := fbInv[i].frozen_s_out;

    // Atualizar p_ref_pct efetivo (drop_comms reduz gradualmente)
    IF g_Inv_CommsDrop[i] THEN
        g_Inv_P_Ref_Pct[i] := fbInv[i].p_ref_pct_out;
    END_IF

END_FOR

// ---------------------------------------------------------------------------
// 3. Agregação no PCC
// ---------------------------------------------------------------------------
p_gen := 0.0;
q_gen := 0.0;
FOR i := 0 TO 17 DO
    p_gen := p_gen + g_Inv_P_kW[i];
    q_gen := q_gen + g_Inv_Q_kVAr[i];
END_FOR
g_P_Gen_Total_kW   := p_gen;
g_Q_Gen_Total_kVAr := q_gen;

// ---------------------------------------------------------------------------
// 4. 1ª iteração Thévenin (tensão com carga nominal)
// ---------------------------------------------------------------------------
p_pcc_0 := load_p0_kw   - p_gen;
q_pcc_0 := load_q0_kvar - q_gen;

fbThevenin(
    p_pcc_kw   := p_pcc_0,
    q_pcc_kvar := q_pcc_0,
    vth_ll_v   := THEVENIN_VTH_LL_V,
    r_ohm      := THEVENIN_R_OHM,
    x_ohm      := THEVENIN_X_OHM
);
v_pcc_0 := fbThevenin.v_pcc_ll_v;

// ---------------------------------------------------------------------------
// 5. Correção ZIP com tensão calculada
// ---------------------------------------------------------------------------
fbZipLoad(
    p0_kw   := load_p0_kw,
    q0_kvar := load_q0_kvar,
    v_ll_v  := v_pcc_0,
    v0_ll_v := V_LL_V,
    a_Z     := ZIP_P_Z,
    a_I     := ZIP_P_I,
    a_P     := ZIP_P_P,
    b_Z     := ZIP_Q_Z,
    b_I     := ZIP_Q_I,
    b_P     := ZIP_Q_P
);
load_p_kw   := fbZipLoad.p_kw;
load_q_kvar := fbZipLoad.q_kvar;

// ---------------------------------------------------------------------------
// 6. 2ª iteração Thévenin (com carga corrigida pelo ZIP)
// ---------------------------------------------------------------------------
p_pcc := load_p_kw   - p_gen;
q_pcc := load_q_kvar - q_gen;

s_pcc_sq := p_pcc * p_pcc + q_pcc * q_pcc;
s_pcc    := SQRT(s_pcc_sq);

fbThevenin(
    p_pcc_kw   := p_pcc,
    q_pcc_kvar := q_pcc,
    vth_ll_v   := THEVENIN_VTH_LL_V,
    r_ohm      := THEVENIN_R_OHM,
    x_ohm      := THEVENIN_X_OHM
);
v_pcc_ll := fbThevenin.v_pcc_ll_v;

// Atualizar grandezas internas do PCC
g_Meter_P_PCC_kW   := p_pcc;
g_Meter_Q_PCC_kVAr := q_pcc;
g_Meter_V_PCC_LL_V := v_pcc_ll;

// ---------------------------------------------------------------------------
// 7. Fator de potência no PCC com sinal
//    Positivo = indutivo (Q_pcc > 0)
//    Negativo = capacitivo (Q_pcc < 0)
// ---------------------------------------------------------------------------
IF s_pcc > 1.0E-9 THEN
    pf_mag := ABS(p_pcc) / s_pcc;
ELSE
    pf_mag := 1.0;
END_IF
IF q_pcc >= 0.0 THEN
    pf_signed := pf_mag;
ELSE
    pf_signed := -pf_mag;
END_IF
g_Meter_PFa := pf_signed;
g_Meter_PFb := pf_signed;
g_Meter_PFc := pf_signed;

// ---------------------------------------------------------------------------
// 8. Tensão no secundário do TP (fase-neutro, V)
//    V_pcc_fn  = V_pcc_ll / sqrt(3)
//    V_mt_fn   = V_pcc_fn × (V_MT_nom / V_BT_nom)
//    V_sec_fn  = V_mt_fn / RTP
// ---------------------------------------------------------------------------
IF v_pcc_ll > 0.0 THEN
    v_pcc_fn := v_pcc_ll * SQRT3_INV;
ELSE
    v_pcc_fn := 0.0;
END_IF

IF V_LL_V > 0.0 THEN
    v_mt_fn  := v_pcc_fn * (V_MT_LL_V / V_LL_V);
ELSE
    v_mt_fn  := 0.0;
END_IF

v_mt_ll  := v_mt_fn * SQRT3;

IF RTP > 0.0 THEN
    v_sec_fn := v_mt_fn / RTP;
ELSE
    v_sec_fn := 0.0;
END_IF

g_Meter_Ua_V := v_sec_fn;
g_Meter_Ub_V := v_sec_fn;
g_Meter_Uc_V := v_sec_fn;

// ---------------------------------------------------------------------------
// 9. Corrente no secundário do TC (A)
//    I_mt_prim = S_pcc / (sqrt(3) × V_mt_ll)
//    I_sec     = I_mt_prim / RTC
// ---------------------------------------------------------------------------
IF v_mt_ll > 0.0 THEN
    i_mt_prim := (s_pcc * 1000.0) / (SQRT3 * v_mt_ll);
ELSE
    i_mt_prim := 0.0;
END_IF

IF RTC > 0.0 THEN
    i_sec := i_mt_prim / RTC;
ELSE
    i_sec := 0.0;
END_IF

g_Meter_Ia_A := i_sec;
g_Meter_Ib_A := i_sec;
g_Meter_Ic_A := i_sec;

// ---------------------------------------------------------------------------
// 10. Codifica grandezas do medidor em registradores U16 para Modbus
// ---------------------------------------------------------------------------
MW_Meter[0]  := FC_EncodePF(g_Meter_PFa);
MW_Meter[1]  := FC_EncodePF(g_Meter_PFb);
MW_Meter[2]  := FC_EncodePF(g_Meter_PFc);
MW_Meter[3]  := 0;
MW_Meter[4]  := 0;
MW_Meter[5]  := 0;
MW_Meter[6]  := 0;
MW_Meter[7]  := FC_EncodeI(g_Meter_Ia_A);
MW_Meter[8]  := FC_EncodeI(g_Meter_Ib_A);
MW_Meter[9]  := FC_EncodeI(g_Meter_Ic_A);
MW_Meter[10] := 0;
MW_Meter[11] := FC_EncodeV(g_Meter_Ua_V);
MW_Meter[12] := FC_EncodeV(g_Meter_Ub_V);
MW_Meter[13] := FC_EncodeV(g_Meter_Uc_V);
MW_Meter[14] := 0;  MW_Meter[15] := 0;  MW_Meter[16] := 0;
MW_Meter[17] := 0;  MW_Meter[18] := 0;  MW_Meter[19] := 0;
MW_Meter[20] := 0;  MW_Meter[21] := 0;  MW_Meter[22] := 0;
MW_Meter[23] := 0;  MW_Meter[24] := 0;  MW_Meter[25] := 0;
MW_Meter[26] := 0;  MW_Meter[27] := 0;

END_FUNCTION_BLOCK

(* ---- FB_Thevenin.st ---- *)
// =============================================================================
// FB_Thevenin — Equivalente de Thévenin (monofásico, referido ao BT)
// Equivalente a TheveninModel em simulation.py
//
// Aproximação linearizada de 1ª ordem:
//   V_pcc_fase ≈ Vth_fase − (R·P_fase + X·Q_fase) / Vth_fase
//
// Convenção P_pcc / Q_pcc:
//   > 0  →  importação da rede  →  tensão cai
//   < 0  →  exportação p/ rede  →  tensão sobe
//
// Parâmetros configurados via GVL_SimConfig (THEVENIN_*).
// =============================================================================

FUNCTION_BLOCK FB_Thevenin
VAR_INPUT
    p_pcc_kw    : REAL;     // Potência ativa no PCC (kW)  + = importa
    q_pcc_kvar  : REAL;     // Potência reativa no PCC (kVAr)
    vth_ll_v    : REAL;     // Tensão de Thévenin LL (V)
    r_ohm       : REAL;     // Resistência equivalente (Ω)
    x_ohm       : REAL;     // Reatância equivalente (Ω)
END_VAR
VAR_OUTPUT
    v_pcc_ll_v  : REAL;     // Tensão linha-linha no PCC (V)
END_VAR
VAR
    vth_fase    : REAL;
    p_fase_w    : REAL;
    q_fase_var  : REAL;
    delta_v     : REAL;
    v_pcc_fase  : REAL;
    SQRT3       : REAL := 1.7320508;
END_VAR

vth_fase := vth_ll_v / SQRT3;

IF vth_fase < 1.0 THEN
    v_pcc_ll_v := 0.0;
    RETURN;
END_IF

p_fase_w    := p_pcc_kw   * 1000.0 / 3.0;
q_fase_var  := q_pcc_kvar * 1000.0 / 3.0;

delta_v     := (r_ohm * p_fase_w + x_ohm * q_fase_var) / vth_fase;
v_pcc_fase  := vth_fase - delta_v;

IF v_pcc_fase < 0.0 THEN v_pcc_fase := 0.0; END_IF

v_pcc_ll_v := v_pcc_fase * SQRT3;

END_FUNCTION_BLOCK

(* ---- FB_ZipLoad.st ---- *)
// =============================================================================
// FB_ZipLoad — Modelo de carga ZIP (coeficientes ANEEL)
// Equivalente a ZipLoadModel em simulation.py
//
// Coeficientes ANEEL para alimentadores de distribuição:
//   P: 50% impedância constante (Z) + 50% potência constante (P)
//   Q: 100% potência constante (P)
//
// Equações:
//   P_load = P0 × (aZ·Vr² + aI·Vr + aP)
//   Q_load = Q0 × (bZ·Vr² + bI·Vr + bP)
//   onde Vr = V_atual / V_nominal
// =============================================================================

FUNCTION_BLOCK FB_ZipLoad
VAR_INPUT
    p0_kw       : REAL;     // Potência ativa nominal da carga (kW)
    q0_kvar     : REAL;     // Potência reativa nominal da carga (kVAr)
    v_ll_v      : REAL;     // Tensão atual linha-linha (V)
    v0_ll_v     : REAL;     // Tensão nominal de referência (V)
    // Coeficientes ZIP para P
    a_Z         : REAL;
    a_I         : REAL;
    a_P         : REAL;
    // Coeficientes ZIP para Q
    b_Z         : REAL;
    b_I         : REAL;
    b_P         : REAL;
END_VAR
VAR_OUTPUT
    p_kw        : REAL;     // Potência ativa ajustada (kW)
    q_kvar      : REAL;     // Potência reativa ajustada (kVAr)
END_VAR
VAR
    vr          : REAL;
    vr2         : REAL;
END_VAR

IF v0_ll_v < 1.0 THEN
    // Proteção divisão por zero — retorna valores nominais
    p_kw  := p0_kw;
    q_kvar := q0_kvar;
    RETURN;
END_IF

vr  := v_ll_v / v0_ll_v;
vr2 := vr * vr;

p_kw   := p0_kw   * (a_Z * vr2 + a_I * vr + a_P);
q_kvar := q0_kvar * (b_Z * vr2 + b_I * vr + b_P);

END_FUNCTION_BLOCK

(* ---- PRG_Main.st ---- *)
// =============================================================================
// PRG_Main — Programa principal do simulador
// Equivalente a main.py (task loop)
//
// Deve ser chamado pela Task Cíclica do Codesys com período = TICK_S (50 ms).
//
// CONFIGURAÇÃO DA TASK no Codesys:
//   Nome    : Task_Simulator
//   Tipo    : Cíclica
//   Período : 50 ms         (coincide com TICK_S = 0.05 s)
//   Prioridade: 2           (abaixo do Modbus, acima do HMI)
//
// MAPEAMENTO MODBUS SLAVE (configurar no Codesys Modbus RTU Slave):
//
//   Porta COM1-A (slave 100, medidor):
//     Holding Registers (FC03): MW_Meter[0..27]
//     Base address: 153 (0x0099)
//
//   Porta COM1-B (slave 101, inversor 0):
//     Holding Registers (FC16): %MW mapeado em g_Inv_P_Ref_Pct[0] e g_Inv_PF_Cmd_Raw[0]
//     HR 256 → g_Inv_P_Ref_Pct[0]   (REAL ou UINT conforme escalonamento)
//     HR 257 → g_Inv_PF_Cmd_Raw[0]  (INT)
//     (ver nota de escalonamento abaixo)
//
//   Porta COM2-A (slave 201, inversor 9):
//     HR 256 → g_Inv_P_Ref_Pct[9]
//     HR 257 → g_Inv_PF_Cmd_Raw[9]
//
//   Porta COM2-B (slave 202, inversor 10):
//     HR 256 → g_Inv_P_Ref_Pct[10]
//     HR 257 → g_Inv_PF_Cmd_Raw[10]
//
// NOTA DE ESCALONAMENTO DO MODBUS:
//   HR 256 (%P): o master escreve 0..100 como UINT. Codesys recebe como UINT.
//   Converter: g_Inv_P_Ref_Pct[i] := UINT_TO_REAL(MW_Inv_P_Raw[i]);
//   HR 257 (FP raw): o master escreve 1..100 como UINT.
//   Converter: g_Inv_PF_Cmd_Raw[i] := UINT_TO_INT(MW_Inv_PF_Raw[i]);
//
//   Se o driver Modbus do Codesys mapear diretamente em variáveis tipadas,
//   ajustar os tipos conforme necessário.
// =============================================================================

PROGRAM PRG_Main
VAR
    fbSim           : FB_Simulator;

    // Registradores raw escritos pelo driver Modbus (UINT, 0-based)
    // Estes são os buffers de recepção do driver Modbus Slave.
    // Mapeados via I/O Mapping do Codesys para as portas RS485.
    //
    // COM1-B: inversor 0 (slave 101)
    MW_Inv_P_Raw    : ARRAY[0..17] OF UINT := [18(0)];  // HR 256 de cada inversor
    MW_Inv_PF_Raw   : ARRAY[0..17] OF UINT := [18(100)]; // HR 257 de cada inversor

    i               : INT;
    bFirstScan      : BOOL := TRUE;
END_VAR

// ===========================================================================
// PRIMEIRA VARREDURA: inicializar modo
// ===========================================================================
IF bFirstScan THEN
    bFirstScan  := FALSE;
    g_SimMode   := SIM_MODE_LOOPBACK;   // Inicia sempre em loopback (Etapa 1)
    g_Reset     := TRUE;                // Limpa estados
END_IF

// ===========================================================================
// COPIAR REGISTRADORES MODBUS → VARIÁVEIS DE SIMULAÇÃO
// Converte UINT (recebido via Modbus) para os tipos internos.
// ===========================================================================
FOR i := 0 TO 17 DO
    // HR 256: setpoint %P (0..100 inteiro)
    g_Inv_P_Ref_Pct[i] := UINT_TO_REAL(MW_Inv_P_Raw[i]);
    // Saturar para garantir faixa válida mesmo se master enviar fora
    IF g_Inv_P_Ref_Pct[i] < 0.0   THEN g_Inv_P_Ref_Pct[i] := 0.0;   END_IF
    IF g_Inv_P_Ref_Pct[i] > 100.0 THEN g_Inv_P_Ref_Pct[i] := 100.0; END_IF

    // HR 257: FP raw (1..100)
    g_Inv_PF_Cmd_Raw[i] := UINT_TO_INT(MW_Inv_PF_Raw[i]);
    // Fora de faixa → unitário (decodificado no FB_InverterDyn)
END_FOR

// ===========================================================================
// EXECUTAR SIMULAÇÃO
// ===========================================================================
fbSim();

// ===========================================================================
// MW_Meter[] é atualizado pelo FB_Simulator e lido automaticamente pelo
// driver Modbus Slave quando o master faz FC03 ao slave 100.
// Nenhuma cópia adicional necessária.
// ===========================================================================

END_PROGRAM
